PROGRAM MAIN
VAR
	
	// Definieren der Prozessparameter
	Param_Menge_Entleeren			:REAL := 10;
	Param_Wartedauer				:TIME := T#10S;
	Param_Haltedauer				:TIME := T#10S;
	Param_Ruehradauer				:TIME := T#10S;
	Param_Ruehrgeschw				:REAL := 10;

	// Instanzierung der Grundfunktionen
	Entleeren		:GF_Entleeren;
	
	CW	:RezeptControlWord;
	
	
END_VAR

Reaktoranlage();
Zuweisung();
Test();

Entleeren.M_START();

CW.CW0 := 4;

END_PROGRAM

(* stored: Version 1.1.0.1, ProductVersion 3.1.4024.12
   POU MAIN: Id {26b9df25-7643-42fb-8a0d-7af5b34d4ed3}, SpecialFunc None *)
